FUNCTION_BLOCK FB_EventF20
VAR_INPUT
	FB_Bacnet : FB_BACnet_DAIKIN_MasterStation_III_No_5;
  	FB_Bacnet_b : FB_BACnet_DAIKIN_MasterStation_III_No_6;
END_VAR
VAR_OUTPUT
	sDebug : STRING(200);
END_VAR
VAR
	fbMsg : FB_TcMessage;
	aUnits : ARRAY[1..21] OF AC_Unit_Status;
	stUnit   : AC_Unit_Status;
	i: INT;
	sMsgText: STRING;

END_VAR
VAR RETAIN
	aPrevState : ARRAY[1..21] OF BOOL := [FALSE(*21*)];
END_VAR

//aUnits[1].bPresVal := FB_Bacnet.StartStopStatus_128.bPresVal;
//aUnits[1].sUnitName := 'F20-A1 (1-00)';
aUnits[2].bPresVal := FB_Bacnet.StartStopStatus_129.bPresVal;
aUnits[2].sUnitName := 'F20-A2 (1-01)';
aUnits[3].bPresVal := FB_Bacnet.StartStopStatus_130.bPresVal;
aUnits[3].sUnitName := 'F20-A3 (1-02)';
aUnits[4].bPresVal := FB_Bacnet.StartStopStatus_131.bPresVal;
aUnits[4].sUnitName := 'F20-A4 (1-03)';
//aUnits[5].bPresVal := FB_Bacnet.StartStopStatus_132.bPresVal;
//aUnits[5].sUnitName := 'F20-B1 (1-04)';
//aUnits[6].bPresVal := FB_Bacnet.StartStopStatus_133.bPresVal;
//aUnits[6].sUnitName := 'F20-B2 (1-05)';
aUnits[7].bPresVal := FB_Bacnet.StartStopStatus_134.bPresVal;
aUnits[7].sUnitName := 'F20-C1 (1-06)';
aUnits[8].bPresVal := FB_Bacnet.StartStopStatus_135.bPresVal;
aUnits[8].sUnitName := 'F20-C2 (1-07)';
aUnits[9].bPresVal := FB_Bacnet.StartStopStatus_136.bPresVal;
aUnits[9].sUnitName := 'F20-D1 (1-08)';
aUnits[10].bPresVal := FB_Bacnet.StartStopStatus_137.bPresVal;
aUnits[10].sUnitName := 'F20-D2 (1-09)';
aUnits[11].bPresVal := FB_Bacnet.StartStopStatus_138.bPresVal;
aUnits[11].sUnitName := 'F20-D3 (1-10)';
aUnits[12].bPresVal := FB_Bacnet.StartStopStatus_139.bPresVal;
aUnits[12].sUnitName := 'F20-D4 (1-11)';
//aUnits[13].bPresVal := FB_Bacnet.StartStopStatus_140.bPresVal;
//aUnits[13].sUnitName := 'F20-E1 (1-12)';
//aUnits[14].bPresVal := FB_Bacnet.StartStopStatus_141.bPresVal;
//aUnits[14].sUnitName := 'F20-E2 (1-13)';
//aUnits[15].bPresVal := FB_Bacnet.StartStopStatus_142.bPresVal;
//aUnits[15].sUnitName := 'F20-E3 (1-14)';
aUnits[16].bPresVal := FB_Bacnet.StartStopStatus_143.bPresVal;
aUnits[16].sUnitName := 'F20-F1 (1-15)';
aUnits[17].bPresVal := FB_Bacnet.StartStopStatus_144.bPresVal;
aUnits[17].sUnitName := 'F20-F2 (2-00)';
//aUnits[18].bPresVal := FB_Bacnet.StartStopStatus_145.bPresVal;
//aUnits[18].sUnitName := 'F20-G1 (2-01)';
//aUnits[19].bPresVal := FB_Bacnet.StartStopStatus_146.bPresVal;
//aUnits[19].sUnitName := 'F20-G2 (2-02)';
aUnits[20].bPresVal := FB_Bacnet.StartStopStatus_147.bPresVal;
aUnits[20].sUnitName := 'F20-H (2-03)';
aUnits[21].bPresVal := FB_Bacnet_b.StartStopStatus_033.bPresVal;
aUnits[21].sUnitName := 'F20-Lobi (3-01)';

FOR i := 1 TO 21 DO
    stUnit := aUnits[i];

    // Detect ON/OFF state change
    IF aUnits[i].bPresVal <> aPrevState[i] THEN
        // --------------------------------------------------------
        // (a) Send TwinCAT message as before
        // --------------------------------------------------------
        IF aUnits[i].bPresVal THEN
            sMsgText := CONCAT(stUnit.sUnitName, ' is Turned ON');
        ELSE
            sMsgText := CONCAT(stUnit.sUnitName, ' is Turned OFF');
        END_IF

        fbMsg.CreateEx(TC_EVENTS.UnitPowerStatus.EventPowerStatus, 0);
        fbMsg.ipArguments.AddString(sMsgText);
        fbMsg.Send(0);

        // --------------------------------------------------------
        // (b) Push event to global CSV queue (for P_CSVWrite_TextMode)
        // --------------------------------------------------------
        IF g_iCount < g_CSV_BUF_SIZE THEN
            g_aUnitName[g_iWriteIdx] := stUnit.sUnitName;
            g_aState[g_iWriteIdx]    := aUnits[i].bPresVal;
            g_iWriteIdx := g_iWriteIdx + 1;
            IF g_iWriteIdx > g_CSV_BUF_SIZE THEN g_iWriteIdx := 1; END_IF
            g_iCount := g_iCount + 1;
        END_IF

        // --------------------------------------------------------
        // (c) Update previous state
        // --------------------------------------------------------
        aPrevState[i] := aUnits[i].bPresVal;
    END_IF
END_FOR

// ------------------------------------------------------------
// Optional debug info
// ------------------------------------------------------------
sDebug := CONCAT('Queued=', INT_TO_STRING(g_iCount));

END_FUNCTION_BLOCK

(* stored: Version 1.1.0.1, ProductVersion 3.1.4024.14
   POU FB_EventF20: Id {6b3d602b-b984-44ff-b4c5-3997f86a9ffa}, SpecialFunc None *)
